FUNCTION_BLOCK EdgeDetection
VAR_INPUT
	In1: BOOL;
END_VAR
VAR_OUTPUT
	out1: BOOL;
END_VAR
VAR
	EdgeDetection1: R_TRIG;
	MemoryCell1: RS;
END_VAR

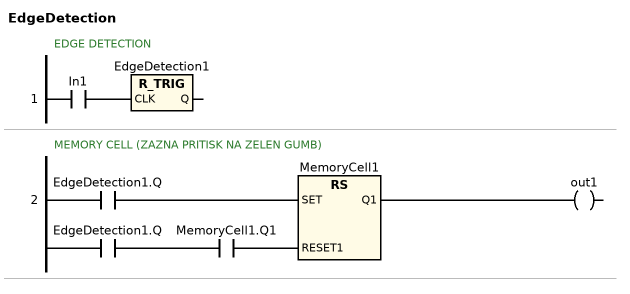
// NETWORK 1
// EDGE DETECTION
EdgeDetection1(CLK := In1); // R_TRIG

// NETWORK 2
// MEMORY CELL (ZAZNA PRITISK NA ZELEN GUMB)
MemoryCell1(SET := EdgeDetection1.Q, RESET1 := EdgeDetection1.Q AND MemoryCell1.Q1); // RS
out1 := MemoryCell1.Q1;

END_FUNCTION_BLOCK

(* stored: Version 1.1.0.1, ProductVersion 3.1.4024.15
   POU EdgeDetection: Id {3d967532-f65e-47b7-be3d-802556be1040}, SpecialFunc None *)
